PROGRAM MAIN
VAR
	bExecute:					BOOL;
	fbFunctionBlock01:		FB_UnitTestTarget01;
	fbFunctionBlock02:		FB_UnitTestTarget02;
END_VAR

// Run
fbTestsuites();

IF bExecute THEN
	bExecute:= NOT fbTestsuites.M_Request(E_Base.Execute);
END_IF

fbFunctionBlock01();
fbFunctionBlock02();

END_PROGRAM

(* stored: Version 1.1.0.1
   POU MAIN: Id {b940f57f-5717-4eac-b98f-4ae3eec6571c}, SpecialFunc None *)
